{attribute 'qualified_only'}
VAR_GLOBAL
	Axis : AXIS_REF;
END_VAR

(* stored: Version 1.1.0.1, ProductVersion 3.1.4024.13
   GVL GVL: Id {e4183608-5164-4b25-a8f1-b40994c935df} *)
